TYPE E_ServerSteps :
(
	SERVER_STATE_IDLE,
	SERVER_STATE_LISTENER_OPEN_START,
	SERVER_STATE_LISTENER_OPEN_WAIT,
	SERVER_STATE_REMOTE_CLIENTS_COMM,
	SERVER_STATE_REMOTE_CLIENTS_CLOSE,
	SERVER_STATE_LISTENER_CLOSE_START,
	SERVER_STATE_LISTENER_CLOSE_WAIT,
	SERVER_STATE_ERROR
);
END_TYPE

(* stored: Version 1.1.0.1, ProductVersion 3.1.4024.3
   DUT E_ServerSteps: Id {c2024b29-2bff-4653-9643-00fbcc18b76b} *)
